Staubli VAL3: call.dtx

mdesc nom_speed = {rmax=9999, blend=off}
